(* PLC project MC3_Multi_IPC1, Beckhoff Automation GmbH TwinCAT PLC Control 3.5.20.30 *)
(* stored: creationDateTime 2025-01-24T10:31:09.1340553, modificationDateTime 2025-01-24T10:31:09.1400543 *)

TYPE ST_XtsCommandFeedback :
STRUCT
		(* Returns wether the execution of the method is done. *)
		IsDone : BOOL;
		(* Returns wether the execution of the method is busy. *)
		IsBusy : BOOL;
		(* Returns wether the execution of the method is busy. *)
		HasError : BOOL;
		(* Returns the HRESULT to the call. *)
		{attribute 'GUID' := '18071995-0000-0000-0000-000000000019'}
		{attribute 'GlobalType'}
		HRESULT : GLOBAL.HRESULT;
	END_STRUCT
END_TYPE

TYPE ST_MoverInfo :
STRUCT

	MoverOtcid :  STRING(20);
	IsVirtuell : BOOL;
	IsActive : BOOL;
	ActPos: LREAL;
	ActVelo: LREAL;
	PlanarMoverCommandMode :STRING(30);// MC_Planar_Mover_Command_Mode;
	State : STRING(20);//MC_Planar_State;
	Positition : LREAL;
	Track :STRING(20);
	Error: BOOL;
	ErrorID : UDINT;
	TargetTrackPosition  : LREAL;
	TargetTrack : Otcid;
	RemainingDistance : LREAL;
	Gap : LREAL;
	LimitVelo : LREAL; 
	LimitAcc : LREAL;
	LimitDec : LREAL;
	LimitJerk : LREAL;
	
END_STRUCT
END_TYPE

TYPE ST_MoverOnTrackInfo :
STRUCT
	TargetPosition 		: LREAL;
	TargetTrack 		: Otcid;
	Remainingdistance 	: LREAL;
	Gap 				: LREAL;
	LimitV 				: LREAL;
	LimitA 				: LREAL;
	LimitD 				: LREAL;
	LimitJ 				: LREAL;
	GapMode				: MC.MC_GAP_MODE_ON_TRACK;
	DynamicMode			: MC.MC_DYNAMIC_MODE_ON_TRACK;
	Movementtype		: MC.MC_MOVEMENT_TYPE_ON_TRACK;
	
END_STRUCT
END_TYPE

INTERFACE I_Mover
METHOD CycleUpdate : BOOL
VAR_INPUT
END_VAR
END_METHOD
METHOD Init : BOOL
VAR_INPUT
	XtsMover:  I_XtsXlMover1;
	XtsProcessingUnit :  I_XtsProcessingUnit1;
END_VAR
END_METHOD
METHOD JoinNearestTrack : BOOL


VAR

END_VAR
END_METHOD
METHOD LeaveSystemAt : BOOL
VAR_INPUT
	ConnectionOut: REFERENCE TO MC_PlanarTrackConnectionOut;	
	gap : LREAL; 		
END_VAR
END_METHOD
METHOD MoveOnTrack : BOOL
VAR_INPUT
	track: REFERENCE TO MC_PlanarTrack;	
	targetPos: LREAL;
	gap : LREAL; 

END_VAR
END_METHOD
METHOD SyncToOtherMover : Bool
VAR_INPUT
	masterSyncPos : LREAL; // Position on the master track
	followerSyncPos : LREAL; // position on the follower track
	PlanarMoverToFollow: REFERENCE TO Tc3_Mc3PlanarMotion.MC_PlanarMover;
	masterTrack : REFERENCE TO Tc3_Mc3PlanarMotion.MC_PlanarTrack; 
	followerTrack : REFERENCE TO Tc3_Mc3PlanarMotion.MC_PlanarTrack; 
	velo :  REFERENCE TO LREAL; 
END_VAR
END_METHOD
METHOD  UpdateXtsTrack
VAR_INPUT
END_VAR
VAR

END_VAR
END_METHOD
PROPERTY distToEndOfTrack : Lreal
END_PROPERTY
PROPERTY MoverStopped : BOOL
END_PROPERTY
PROPERTY P_Dynamics : REFERENCE TO DynamicConstraint_PathXY;
END_PROPERTY
PROPERTY P_IsInitialized : bool
END_PROPERTY
PROPERTY P_MoverOTCID : OTCID
END_PROPERTY
PROPERTY P_PlanarFeedback : REFERENCE TO MC_PlanarFeedback
END_PROPERTY
PROPERTY P_PlanarMover :   REFERENCE TO  MC_PlanarMover
END_PROPERTY
PROPERTY P_SyncFeedback :  REFERENCE TO MC_PlanarFeedbackGearInPosOnTrackWithMasterMover
END_PROPERTY
PROPERTY P_TargetTrack : UDINT
END_PROPERTY
PROPERTY Rework : BOOL
END_PROPERTY
PROPERTY XlProcessingUnit : I_XtsProcessingUnit1
END_PROPERTY
PROPERTY XtsComFeed : REFERENCE TO  XtsCommandFeedback
END_PROPERTY
PROPERTY XtsXlMover :  I_XtsXlMover1
END_PROPERTY
END_INTERFACE

{attribute 'no_assign'}
FUNCTION_BLOCK FB_Mover IMPLEMENTS I_Mover
VAR_INPUT
END_VAR
VAR_OUTPUT
END_VAR
VAR
	_bIsInitialized: BOOL;	

	fbPlanarMover : MC_PlanarMover;
	fbPlanarFeedback: MC_PlanarFeedback;
	trackTrail: MC_PlanarTrackTrail;
	SyncMoverFeedback: Tc3_Mc3PlanarMotion.MC_PlanarFeedbackGearInPosOnTrackWithMasterMover;
	
	_GearInOptions: Tc3_Mc3PlanarMotion.ST_GearInPosOnTrackWithMasterMoverOptions;
	_stMoveOnTrackOptions: ST_MoveOnTrackOptions;
	_stLeaveSystemAtOptions : ST_LeaveSystemAtOptions;
	
	_syncTrail : MC_PlanarTrackTrail;
	
	CmdFeedback :  XtsCommandFeedback;
	ipXtsMover:   I_XtsXlMover1;
	ipXtsProcessingUnit:  I_XtsProcessingUnit1;

	_stMoverInfos : ST_MoverInfo;	
	_stMoverOnTrackInfos : ST_MoverOnTrackInfo;

	_nextMcTrackOid: OTCID;
	_stDynamics: DynamicConstraint_PathXY;
	_TargetTrack : UDINT;
	_ReWork : BOOL;
	_partConfig: UINT;
	_InSync :BOOL; 
	_PositionOnTrack : LREAL;
	_Track : OTCID; 
	_distToEndOfTrack : LREAL;

	fbResult						: FB_TcMessage;
	_ipComObject					: ITComObject;
	PID_OnTrackInfos				: PTCID := 16#05030180;
	bInit 							: BOOL;
END_VAR

            
          

METHOD CycleUpdate : BOOL
VAR_INPUT
END_VAR

VAR_INST
	_trackEnum: e_TrackNum;

END_VAR
                  IF NOT _bIsInitialized THEN
	RETURN;
END_IF

fbPlanarMover.GetTrackTrailInformation(trackTrail);
_PositionOnTrack := fbPlanarMover.MCTOPLC.SETONTRACK.SetPos;
IF fbPlanarMover.MCTOPLC.SETONTRACK.TrackOID<>0 THEN 
	_Track := fbPlanarMover.MCTOPLC.SETONTRACK.TrackOID;
	_trackEnum := F_GetTrackEnum(fbPlanarMover.MCTOPLC.SETONTRACK.TrackOID); 
	_distToEndOfTrack := GVL_Mc.aMCTracks[_trackEnum].GetLength()-_PositionOnTrack;
END_IF

fbPlanarMover.Update();
fbPlanarFeedback.Update();
SyncMoverFeedback.Update();

_stMoverinfos.MoverOtcid :=TO_STRING(fbPlanarMover.MCTOPLC.STD.MoverOID) ;
_stMoverinfos.IsActive := ipXtsMover.GetIsActive(0);
_stMoverinfos.ActPos :=  ipXtsMover.GetPositionInfo_trackPosition(0);
_stMoverinfos.ActVelo := fbPlanarMover.MCTOPLC.SETONTRACK.SetVelo;
_stMoverinfos.IsVirtuell := ipXtsMover.GetIsVirtualFeedbackEnabled(0);
_stMoverinfos.Positition :=	fbPlanarMover.MCTOPLC.SETONTRACK.SetPos;
_stMoverinfos.Track := TO_STRING(_trackEnum);
_stMoverinfos.Error := fbPlanarMover.Error;
_stMoverinfos.ErrorID := fbPlanarMover.ErrorId;
_stMoverinfos.PlanarMoverCommandMode :=  TO_STRING(fbPlanarMover.MCTOPLC.STD.CommandMode);
_stMoverinfos.State :=  TO_STRING(fbPlanarMover.MCTOPLC.STD.State);
_stMoverinfos.Gap := _stMoverOnTrackInfos.Gap;
_stMoverinfos.LimitAcc := _stMoverOnTrackInfos.LimitA;
_stMoverinfos.LimitDec := _stMoverOnTrackInfos.LimitD;
_stMoverinfos.LimitJerk := _stMoverOnTrackInfos.LimitJ;
_stMoverinfos.LimitVelo := _stMoverOnTrackInfos.LimitV;
_stMoverinfos.TargetTrackPosition := _stMoverOnTrackInfos.TargetPosition;
_stMoverinfos.TargetTrack := _stMoverOnTrackInfos.TargetTrack;
_stMoverinfos.RemainingDistance := _stMoverOnTrackInfos.Remainingdistance;




UpdateXtsTrack();
GetOnTrackInfos() ;




                
END_METHOD

METHOD GetComObject : BOOL
VAR_INPUT
	nObjectId: OTCID;
END_VAR
                  IF FW_ObjMgr_GetObjectInstance(	oid		:= nObjectId, 
								iid		:= TC_GLOBAL_IID_LIST.IID_ITComObject, 
								pipUnk	:= ADR(_ipComObject)) = 0
THEN
	GetComObject := TRUE;
END_IF
                
END_METHOD

METHOD GetOnTrackInfos : BOOL
VAR
	nData 			: UDINT := SIZEOF(_stMoverOnTrackInfos);
	pData 			: PVOID := ADR(_stMoverOnTrackInfos);
	stEventEntry	: TcEventEntry;
	pstEventEntry	: REFERENCE TO TcEventEntry REF= stEventEntry;
END_VAR
VAR_INST
	hResult : HRESULT;
	bError : BOOL;
END_VAR
                  bError := FALSE;

IF _ipComObject <> 0 THEN 
	 hResult := 	_ipComObject.TcgetObjPara(		pid := PID_OnTrackInfos,
													nData := nData,
													pData := pData,
													pgp := 0); 	
	IF hResult = 0 THEN
		GetOnTrackInfos := TRUE;
ELSE
	HRESULTAdsErr_TO_TcEventEntry(hResult,stEventEntry);
	IF NOT fbResult.EqualsToEventEntryEx( stOther := stEventEntry) THEN
		fbResult.CreateEx(stEventEntry, 0);
		fbResult.Send(0);
		fbResult.Release();
	END_IF
		bError := TRUE;
	END_IF							
END_IF

                
END_METHOD

METHOD Init : BOOL
VAR_INPUT

	XtsMover:   I_XtsXlMover1;
	XtsProcessingUnit :  I_XtsProcessingUnit1;
END_VAR
                  


ipXtsMover:= XtsMover;
ipXtsProcessingUnit :=  XtsProcessingUnit;

_stMoveOnTrackOptions.direction := MC_Direction.mcDirectionPositive;
_stMoveOnTrackOptions.gapMode := MC_GAP_MODE_ON_TRACK.Fast1D;
_stMoveOnTrackOptions.gap:= 800;

_syncTrail.AddTrack(track:= GVL_Mc.aMCTracks[E_TrackNum.Small]); 
_syncTrail.AddTrack(track:= GVL_Mc.aMCTracks[E_TrackNum.MainStart]); 


//_stDynamics.SetValuesVADJ(500, 4000, 4000, 10000);




	_bIsInitialized := TRUE;
	Init := TRUE;

IF NOT bInit THEN
	IF GetComObject(nObjectId:=fbPlanarMover.MCTOPLC.STD.MoverOID) THEN
		bInit:=TRUE;
	END_IF
	RETURN;
END_IF


                
END_METHOD

METHOD JoinNearestTrack : BOOL


VAR_INST
	nForCounter: UINT;
	mcTrackOid: OTCID;
	partOid: OTCID;
	cmdFeedback					: 	XtsCommandFeedback;
	objectInfo: PlanarObjectInfo;
END_VAR
                  partOid := ipXtsMover.GetPositionInfo_partObjectId(cmdFeedback);

IF partOid = 0 THEN
	RETURN;
END_IF

IF cmdFeedback.IsDone THEN
	mcTrackOid := ipXtsProcessingUnit.XlPartWithOid(partOid, cmdFeedback).GetMcTrackOid(cmdFeedback);
	
	FOR nForCounter := 1 TO GVL_MC.nNumTracks DO
		objectInfo := GVL_MC.aMcTracks[nForCounter].GetPlanarObjectInfo();
		IF objectInfo.Id = mcTrackOid THEN
			fbPlanarMover.JoinTrack(fbPlanarFeedback, GVL_MC.aMcTracks[nForCounter], _stDynamics, 0); 
			RETURN;
		END_IF
	END_FOR
END_IF
                
END_METHOD

METHOD LeaveSystemAt : BOOL
VAR_INPUT
	ConnectionOut: REFERENCE TO MC_PlanarTrackConnectionOut;
	gap : LREAL; 
END_VAR
                  _stLeaveSystemAtOptions.gap := gap;
_stLeaveSystemAtOptions.gapMode := MC_GAP_MODE_ON_TRACK.Fast1D; 
_stLeaveSystemAtOptions.dynamicMode :=  MC_DYNAMIC_MODE_ON_TRACK.None;

fbPlanarMover.LeaveSystemAt(fbPlanarFeedback, ConnectionOut,  _stDynamics,_stLeaveSystemAtOptions);

                
END_METHOD

METHOD MoveOnTrack : BOOL
VAR_INPUT
	track: REFERENCE TO MC_PlanarTrack;	
	targetPos: LREAL;
	gap : LREAL; 
END_VAR
                  _stMoveonTrackOptions.gap := gap; 

fbPlanarMover.MoveOnTrack(
	commandFeedback:= fbPlanarFeedback, 
	targetTrack:= track, 
	targetPositionOnTrack:= targetPos, 
	constraint:= _stDynamics, 
	options:= _stMoveOnTrackOptions);
                
END_METHOD

METHOD SyncToOtherMover : BOOL
VAR_INPUT
	masterSyncPos : LREAL; // Position on the master track
	followerSyncPos : LREAL; // position on the follower track
	PlanarMoverToFollow: REFERENCE TO Tc3_Mc3PlanarMotion.MC_PlanarMover;
	masterTrack : REFERENCE TO Tc3_Mc3PlanarMotion.MC_PlanarTrack; 
	followerTrack : REFERENCE TO Tc3_Mc3PlanarMotion.MC_PlanarTrack; 
	velo : REFERENCE TO LREAL; 
END_VAR

VAR
	trail: Tc3_Mc3PlanarMotion.MC_PlanarTrackTrail;

END_VAR
                  _GearInOptions.allowedSlaveSyncDirections := MC_SYNC_DIRECTIONS.Positive; 
_GearInOptions.directionMasterSyncPosition := MC_DIRECTION.mcDirectionNonModulo; 
_GearInOptions.directionSlaveSyncPosition := MC_DIRECTION.mcDirectionNonModulo;  
_GearInOptions.followMover := FALSE; 
_GearInOptions.gap := 0; // elimnate gap funciton 
_GearInOptions.inSyncToleranceDistance :=0; 
_GearInOptions.moduloToleranceMasterSyncPosition := 0; 
_GearInOptions.moduloToleranceSlaveSyncPosition := 0;  
_stDynamics.V := velo; 

fbPlanarMover.GearInPosOnTrackWithMasterMover(
	commandFeedback:=  SyncMoverFeedback , 
	masterMover:= PlanarMoverToFollow , 
	trackTrail:= _syncTrail, // may need to give a trail maybe not
	masterSyncPosition:= masterSyncPos, 
	masterSyncPositionTrack:= MasterTrack , 
	slaveSyncPosition:= followerSyncPos, 
	slaveSyncPositionTrack:= followerTrack, 
	constraint:=_stDynamics , 
	options:=_GearInOptions );
	
                
END_METHOD

METHOD PUBLIC UpdateXtsTrack
VAR_INPUT
END_VAR
VAR_STAT
	nTrackCount: UINT;
	oid1: OTCID;
	oid2: OTCID;
	
	nForCounter: UINT;
	nPartConfigCount: UINT;
	
	partConfig1: OTCID;
	partConfig2: OTCID;
	
	mcTrackOid1: OTCID;
	mcTrackOid2: OTCID;
	trackOid: OTCID;
	
	nTrackTrailCount: UDINT;
	actTrackOid: OTCID;
	nIndexInTrail: UDINT;
END_VAR
                  nTrackTrailCount := trackTrail.TrackCount;
actTrackOid := fbPlanarMover.MCTOPLC.SETONTRACK.TrackOID;

IF nTrackTrailCount <= 1 THEN
	RETURN;
END_IF

FOR nForCounter := 1 TO UDINT_TO_UINT(nTrackTrailCount) DO
	oid1 := trackTrail.GetTrackOidAt(nForCounter);
	IF oid1 = actTrackOid THEN
		IF nForCounter < nTrackTrailCount THEN
			oid2 := trackTrail.GetTrackOidAt(nForCounter + 1);
			EXIT;
		ELSE
			RETURN; //last one ine track trail
		END_IF
	END_IF
END_FOR

IF oid2 = _nextMcTrackOid AND ipXtsMover.GetPositionInfo_partPosition(CmdFeedback) < 600 THEN //no change
	RETURN;
END_IF

nTrackCount := ipXtsProcessingUnit.TrackCount();

FOR nForCounter := 1 TO nTrackCount DO
	nPartConfigCount := ipXtsProcessingUnit.Track(nForCounter, CmdFeedback).PartConfigCount(); 
	
	IF nPartConfigCount >= 2  THEN
		partConfig1 := ipXtsProcessingUnit.Track(nForCounter, CmdFeedback).GetPartConfigOidAt(1, 0);
		partConfig2 := ipXtsProcessingUnit.Track(nForCounter, CmdFeedback).GetPartConfigOidAt(2, 0);
//
		
		IF partConfig1 = 0 OR partConfig2 = 0 THEN
			CONTINUE;
		END_IF
		
		mcTrackOid1 := ipXtsProcessingUnit.XlPartWithOid(partConfig1, CmdFeedback).GetMcTrackOid(0);
		mcTrackOid2 := ipXtsProcessingUnit.XlPartWithOid(partConfig2, CmdFeedback).GetMcTrackOid(0);
		IF mcTrackOid1 = oid1 AND mcTrackOid2 = oid2   THEN
			trackOid := ipXtsProcessingUnit.Track(nForCounter, CmdFeedback).GetObjectId();
			ipXtsMover.SetActiveTrackObjectId(trackOid, CmdFeedback);
			
			IF CmdFeedback.IsDone THEN
				_nextMcTrackOid := oid2;
			END_IF
			
			RETURN;
		END_IF
	END_IF
END_FOR


                
END_METHOD

PROPERTY distToEndOfTrack : Lreal
GET
VAR
END_VAR
                    distToEndOfTrack := _distToEndOfTrack;
                  
END_GET
END_PROPERTY

PROPERTY MoverStopped : BOOL
GET
VAR
END_VAR
                    MoverStopped := (fbPlanarMover.MCTOPLC.SETONTRACK.SetVelo < 20);


                  
END_GET
SET
VAR
END_VAR
                    
                  
END_SET
END_PROPERTY

PROPERTY P_Dynamics : REFERENCE TO DynamicConstraint_PathXY;
GET
VAR
END_VAR
                    
P_Dynamics REF= _stDynamics; 
                  
END_GET
END_PROPERTY

PROPERTY P_IsInitialized : bool
GET
VAR
END_VAR
                    P_IsInitialized := _bIsInitialized;
                  
END_GET
END_PROPERTY

PROPERTY P_MoveOnTrackOptions  : REFERENCE TO  ST_MoveOnTrackOptions
GET
VAR
END_VAR
                    P_MoveOnTrackOptions REF= _stMoveOnTrackOptions;
                  
END_GET
END_PROPERTY

PROPERTY P_MoverInfos : REFERENCE TO ST_MoverInfo
GET
VAR
END_VAR
                    P_MoverInfos  REF= _stMoverInfos;
                  
END_GET
END_PROPERTY

PROPERTY p_MoverOTCID : OTCID
GET
VAR
END_VAR
                    p_MoverOTCID := fbPlanarMover.MCTOPLC.STD.MoverOID;
                  
END_GET
SET
VAR
END_VAR
                    
                  
END_SET
END_PROPERTY

PROPERTY P_PlanarFeedback : REFERENCE TO MC_PlanarFeedback
GET
VAR
END_VAR
                    P_PlanarFeedback REF= fbPlanarFeedback;
                  
END_GET
END_PROPERTY

PROPERTY P_PlanarMover :   REFERENCE TO  MC_PlanarMover
GET
VAR
END_VAR
                    P_PlanarMover REF= fbPlanarMover;
                  
END_GET
END_PROPERTY

PROPERTY P_SyncFeedback :  REFERENCE TO MC_PlanarFeedbackGearInPosOnTrackWithMasterMover
GET
VAR
END_VAR
                    P_SyncFeedback REF= SyncMoverFeedback; 
                  
END_GET
END_PROPERTY

PROPERTY P_TargetTrack : UDINT
GET
VAR
END_VAR
                    P_TargetTrack := _TargetTrack ;
                  
END_GET
SET
VAR
END_VAR
                    _TargetTrack := P_TargetTrack; 
                  
END_SET
END_PROPERTY

PROPERTY Rework : BOOL
GET
VAR
END_VAR
                    Rework := _Rework;

                  
END_GET
SET
VAR
END_VAR
                    _Rework := Rework;
                  
END_SET
END_PROPERTY

PROPERTY XlProcessingUnit : I_XtsProcessingUnit1
GET
VAR
END_VAR
                    XlProcessingUnit := ipXtsProcessingUnit;
                  
END_GET
END_PROPERTY

PROPERTY XtsComFeed : REFERENCE TO  XtsCommandFeedback
GET
VAR
END_VAR
                    XtsComFeed REF= CmdFeedback;
                  
END_GET
END_PROPERTY

PROPERTY XtsXlMover : I_XtsXlMover1
GET
VAR
END_VAR
                    XtsXlMover := ipXtsMover;
                  
END_GET
END_PROPERTY
END_FUNCTION_BLOCK
